{attribute 'OPC.UA.DA.StructuredType' := '1'}
	{attribute 'OPC.UA.DA' := '1'}
TYPE ST_GripperSpecific :
STRUCT

END_STRUCT
END_TYPE

(* stored: Version 1.1.0.1, ProductVersion 3.1.4026.18
   DUT ST_GripperSpecific: Id {160838c9-eb4f-4005-8e3e-1344d5051a0c} *)
